PROGRAM Notes
VAR
END_VAR

(*
Har implementert følgende:
- Modbus RTU read og write registers program
- Versjonskontroll/Git
- Har opprettet HMI prosjekt for å vise register verdier
- Spesifisere hva dette programmet skal kunne gjøre
- Sjekke om det finnes allerede eksisterende blokker som har funksjonaliteten jeg ønsker
- Spesifiser hvordan HMI skal se ut

Videre oppgaver:
- Prøve å gå tilbake til en eldre versjon ved hjelp av Git. Lag eget prosjekt for dette
- Implementere bibliotek for testing av funksjonsblokker/TcUnit
- Lage eget bibliotek for egne implementerte funksjonsblokker som er testet med TcUnit




*)

END_PROGRAM

(* stored: Version 1.1.0.1, ProductVersion 3.1.4024.13
   POU Notes: Id {d0b44e49-92c0-4d27-89dd-1d1622b8c00c}, SpecialFunc None *)
